{attribute 'GeneratedUsingTerminal: KL6224-0001'}
{attribute addProperty BoxType "KL6224-0001"}
{attribute addProperty Id "Channel_1AT %Q*Channel_085338040"}
{attribute addProperty CRC "4229837715"}
{attribute addProperty Size "0"}
TYPE KL_FC1E3393 :
STRUCT
	{attribute addProperty Name "Channel_1"}
	Channel_1 : Channel_08533804;
END_STRUCT
END_TYPE

(* stored: Version 1.2.0.0, ProductVersion 3.1.4024.9
   DUT KL_FC1E3393: Id {cd9952cf-11f8-44fe-a77c-a1b39b39d0b1} *)
